% RSLogix 500 project Q1.RSS, saved by version 8.30.00.16 %
PROJECT "Q1"    % processor: Bul.1763 MicroLogix 1100 Series B %

PROGRAM FILES
  LAD 2   6 rungs

DATA FILES
  O0 OUTPUT  4 elements
  I1 INPUT  6 elements
  S2 STATUS  66 elements
  B3 BINARY  1 elements
  T4 TIMER  1 elements
  C5 COUNTER  1 elements
  R6 CONTROL  1 elements
  N7 INTEGER  1 elements
  F8 FLOAT  1 elements

LADDER 2
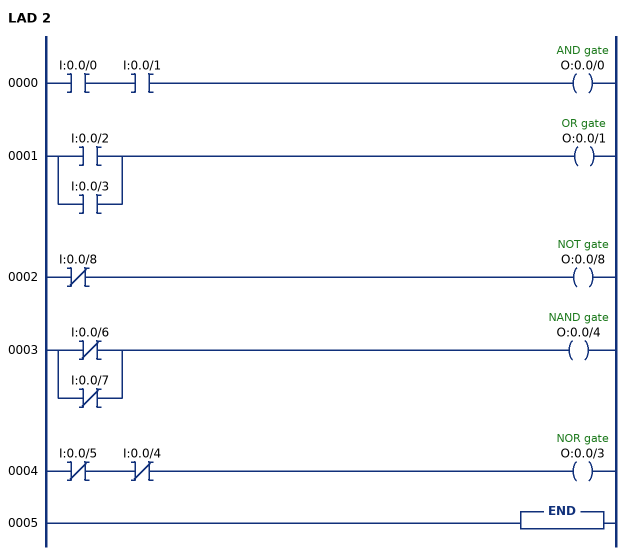
% Rung: 0 %
SOR XIC I:0.0/0 XIC I:0.0/1 OTE O:0.0/0 EOR
%   O:0.0/0  "AND gate" %
% Rung: 1 %
SOR BST XIC I:0.0/2 NXB XIC I:0.0/3 BND OTE O:0.0/1 EOR
%   O:0.0/1  "OR gate" %
% Rung: 2 %
SOR XIO I:0.0/8 OTE O:0.0/8 EOR
%   O:0.0/8  "NOT gate" %
% Rung: 3 %
SOR BST XIO I:0.0/6 NXB XIO I:0.0/7 BND OTE O:0.0/4 EOR
%   O:0.0/4  "NAND gate" %
% Rung: 4 %
SOR XIO I:0.0/5 XIO I:0.0/4 OTE O:0.0/3 EOR
%   O:0.0/3  "NOR gate" %
% Rung: 5 %
SOR END EOR
